(* IEC 61131-3 sources: can_commsgen/tests/golden/plc, 9 files *)

(* ---- DriveMode.st ---- *)
(* THIS FILE IS AUTO-GENERATED. DO NOT EDIT. *)
{attribute 'qualified_only'}
{attribute 'strict'}
TYPE DriveMode : (
    IDLE     := 0,
    VELOCITY := 1,
    POSITION := 2,
    TORQUE   := 3
) USINT;
END_TYPE

(* ---- GVL.gvl.st ---- *)
(* THIS FILE IS AUTO-GENERATED. DO NOT EDIT. *)
{attribute 'qualified_only'}
VAR_GLOBAL
    (* motor_command -- 0x00000100, pc_to_plc *)
    targetVelocity_rpm        : REAL;
    torqueLimit_Nm            : REAL;
    motorCommandWithinTimeout : BOOL;

    (* pc_state -- 0x00000300, pc_to_plc *)
    driveMode                 : DriveMode;
    pcStateWithinTimeout      : BOOL;
END_VAR

(* ---- CAN_EXTRACT_BITS.st ---- *)
(* THIS FILE IS AUTO-GENERATED. DO NOT EDIT. *)
FUNCTION CAN_EXTRACT_BITS : LINT
VAR_INPUT
    data      : ARRAY[0..7] OF USINT;
    bitOffset : UINT;
    bitCount  : UINT;
    signed    : BOOL;
END_VAR
VAR
    i       : UINT;
    byteIdx : UINT;
    bitIdx  : UINT;
    raw     : ULINT;
END_VAR

// --- BEGIN IMPLEMENTATION ---

raw := 0;
FOR i := 0 TO bitCount - 1 DO
    byteIdx := (bitOffset + i) / 8;
    bitIdx  := (bitOffset + i) MOD 8;
    IF (data[byteIdx] AND SHL(USINT#1, bitIdx)) <> 0 THEN
        raw := raw OR SHL(ULINT#1, i);
    END_IF
END_FOR

IF signed AND (raw AND SHL(ULINT#1, bitCount - 1)) <> 0 THEN
    raw := raw OR NOT (SHL(ULINT#1, bitCount) - 1);
END_IF

CAN_EXTRACT_BITS := ULINT_TO_LINT(raw);

(* ---- CAN_INSERT_BITS.st ---- *)
(* THIS FILE IS AUTO-GENERATED. DO NOT EDIT. *)
FUNCTION CAN_INSERT_BITS : BOOL
VAR_INPUT
    value     : LINT;
    bitOffset : UINT;
    bitCount  : UINT;
END_VAR
VAR_IN_OUT
    data      : ARRAY[0..7] OF USINT;
END_VAR
VAR
    i       : UINT;
    byteIdx : UINT;
    bitIdx  : UINT;
    raw     : ULINT;
END_VAR

// --- BEGIN IMPLEMENTATION ---

raw := LINT_TO_ULINT(value);
FOR i := 0 TO bitCount - 1 DO
    byteIdx := (bitOffset + i) / 8;
    bitIdx  := (bitOffset + i) MOD 8;
    IF (raw AND SHL(ULINT#1, i)) <> 0 THEN
        data[byteIdx] := data[byteIdx] OR SHL(USINT#1, bitIdx);
    ELSE
        data[byteIdx] := data[byteIdx] AND NOT SHL(USINT#1, bitIdx);
    END_IF
END_FOR

CAN_INSERT_BITS := TRUE;

(* ---- DriveMode_FROM_INT.st ---- *)
(* THIS FILE IS AUTO-GENERATED. DO NOT EDIT. *)
FUNCTION DriveMode_FROM_INT : DriveMode
VAR_INPUT
    value : USINT;
END_VAR

// --- BEGIN IMPLEMENTATION ---

CASE value OF
    0: DriveMode_FROM_INT := DriveMode.IDLE;
    1: DriveMode_FROM_INT := DriveMode.VELOCITY;
    2: DriveMode_FROM_INT := DriveMode.POSITION;
    3: DriveMode_FROM_INT := DriveMode.TORQUE;
ELSE
    DriveMode_FROM_INT := DriveMode.IDLE;
END_CASE

(* ---- DRIVE_STATUS_SEND.st ---- *)
(* THIS FILE IS AUTO-GENERATED. DO NOT EDIT. *)
FUNCTION_BLOCK DRIVE_STATUS_SEND
VAR_INPUT
    channel            : ifmDevice.CAN_CHANNEL;
    actualVelocity_rpm : REAL;
    motorTemp_degC     : REAL;
    busVoltage_V       : REAL;
    faultCode          : USINT;
END_VAR
VAR
    tx   : ifmRCAN.CAN_Tx;
    data : ARRAY[0..7] OF USINT := [0, 0, 0, 0, 0, 0, 0, 0];
END_VAR

// --- BEGIN IMPLEMENTATION ---

CAN_INSERT_BITS(TO_LINT(REAL_TO_INT(actualVelocity_rpm / 0.1)),  0,  16, data);
CAN_INSERT_BITS(TO_LINT(REAL_TO_INT(motorTemp_degC / 0.1)),       16, 12, data);
CAN_INSERT_BITS(TO_LINT(REAL_TO_UINT(busVoltage_V / 0.1)),        28, 10, data);
CAN_INSERT_BITS(TO_LINT(faultCode),                                38, 8,  data);

tx(xEnable := TRUE, eChannel := channel, xExtended := TRUE,
   udiID := 16#00000200, usiDLC := 6, aData := data);

(* ---- MOTOR_COMMAND_RECV.st ---- *)
(* THIS FILE IS AUTO-GENERATED. DO NOT EDIT. *)
FUNCTION_BLOCK MOTOR_COMMAND_RECV
VAR_INPUT
    channel : ifmDevice.CAN_CHANNEL;
END_VAR
VAR
    rx     : ifmRCAN.CAN_Rx;
    timer  : TON;
    rxData : ARRAY[0..7] OF USINT;
END_VAR

// --- BEGIN IMPLEMENTATION ---

rx(xEnable := TRUE, eChannel := channel, xExtended := TRUE, udiID := 16#00000100);

IF rx.uiAvailable > 0 AND rx.usiDLC = 4 THEN
    rxData := rx.aData;
    GVL.targetVelocity_rpm := TO_REAL(CAN_EXTRACT_BITS(rxData, 0, 16, TRUE)) * 0.1;
    GVL.torqueLimit_Nm     := TO_REAL(CAN_EXTRACT_BITS(rxData, 16, 16, FALSE)) * 0.01;
    timer(IN := FALSE);
END_IF

timer(IN := TRUE, PT := T#500ms);
GVL.motorCommandWithinTimeout := NOT timer.Q;

(* ---- PC_STATE_RECV.st ---- *)
(* THIS FILE IS AUTO-GENERATED. DO NOT EDIT. *)
FUNCTION_BLOCK PC_STATE_RECV
VAR_INPUT
    channel : ifmDevice.CAN_CHANNEL;
END_VAR
VAR
    rx     : ifmRCAN.CAN_Rx;
    timer  : TON;
    rxData : ARRAY[0..7] OF USINT;
END_VAR

// --- BEGIN IMPLEMENTATION ---

rx(xEnable := TRUE, eChannel := channel, xExtended := TRUE, udiID := 16#00000300);

IF rx.uiAvailable > 0 AND rx.usiDLC = 1 THEN
    rxData := rx.aData;
    GVL.driveMode := DriveMode_FROM_INT(TO_USINT(CAN_EXTRACT_BITS(rxData, 0, 2, FALSE)));
    timer(IN := FALSE);
END_IF

timer(IN := TRUE, PT := T#1000ms);
GVL.pcStateWithinTimeout := NOT timer.Q;

(* ---- CAN_RECV.st ---- *)
(* THIS FILE IS AUTO-GENERATED. DO NOT EDIT. *)
PROGRAM CAN_RECV
VAR
    fbMOTOR_COMMAND_RECV : MOTOR_COMMAND_RECV;
    fbPC_STATE_RECV      : PC_STATE_RECV;
END_VAR

// --- BEGIN IMPLEMENTATION ---

fbMOTOR_COMMAND_RECV(channel := ifmDevice.CAN_CHANNEL.CHAN_0);
fbPC_STATE_RECV(channel := ifmDevice.CAN_CHANNEL.CHAN_0);
